// TIA Portal V19 export
FUNCTION "FC_EM_Loading" : Void   // FC3, FBD
{ S7_Optimized_Access := 'TRUE' }
// stored: SetENOAutomatically false
BEGIN

REGION Network 1: ------------------------------------------------------------------------ Inputs ------------------------------------------------------------------------
END_REGION

REGION Network 2: Verwerken iLoadingSenDown_a1
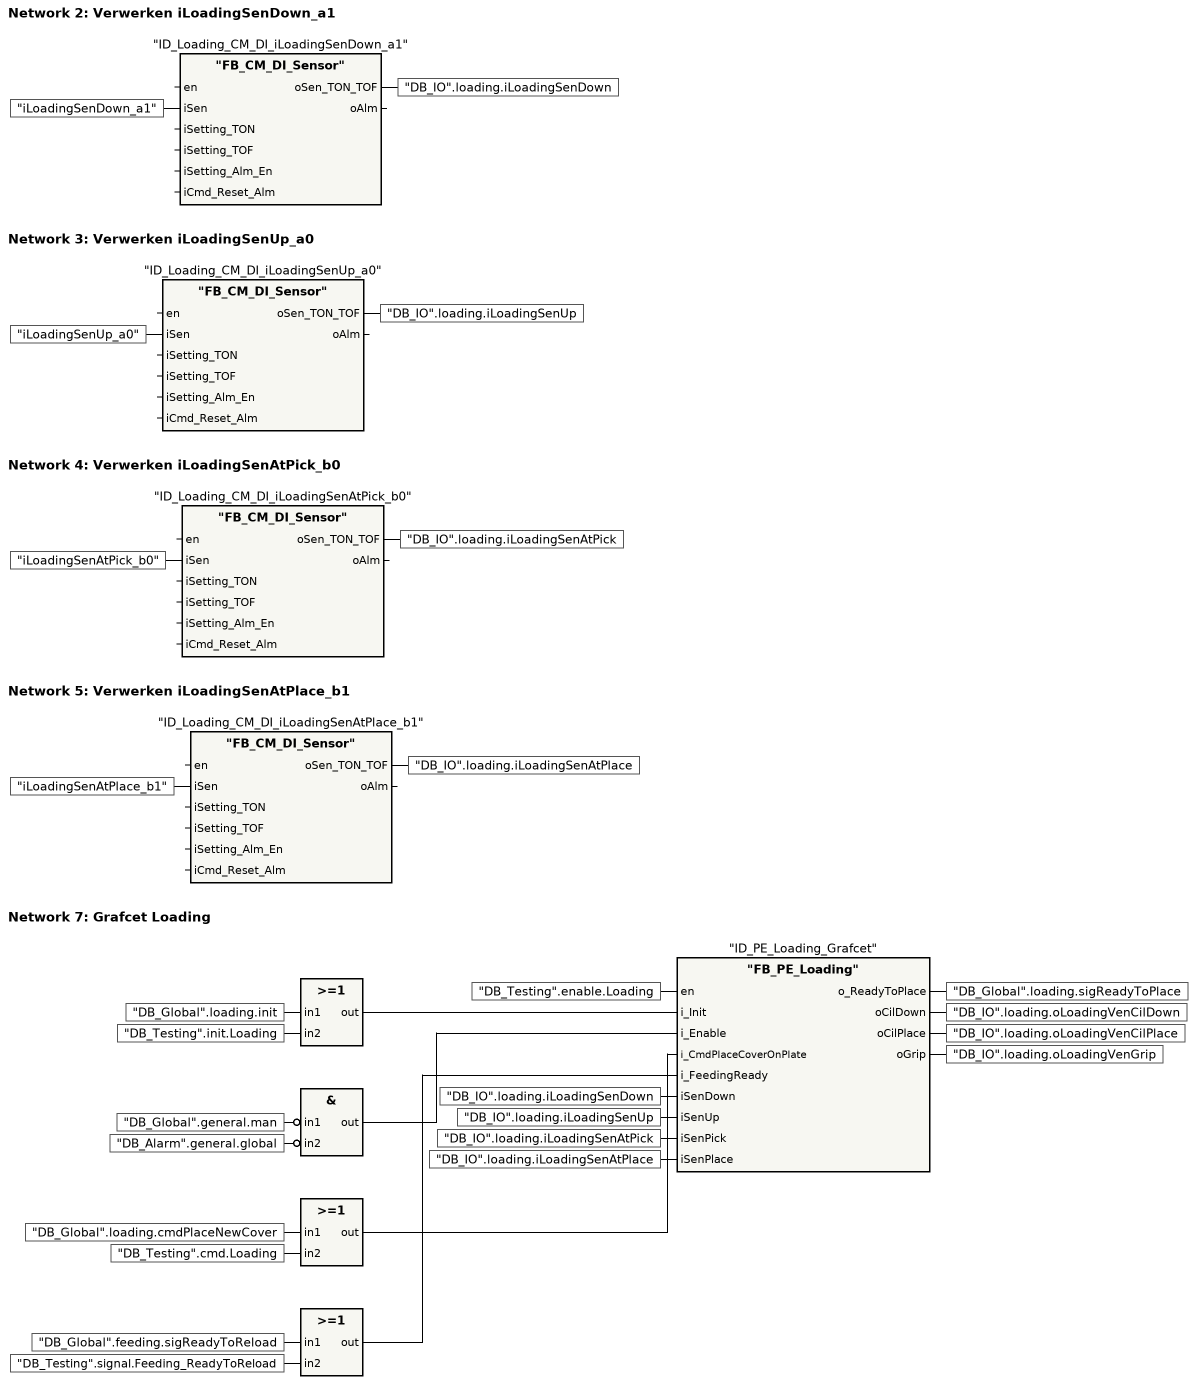
   "ID_Loading_CM_DI_iLoadingSenDown_a1"(iSen := "iLoadingSenDown_a1",   // "FB_CM_DI_Sensor"
                           oSen_TON_TOF => "DB_IO".loading.iLoadingSenDown);
END_REGION

REGION Network 3: Verwerken iLoadingSenUp_a0
   "ID_Loading_CM_DI_iLoadingSenUp_a0"(iSen := "iLoadingSenUp_a0",   // "FB_CM_DI_Sensor"
                           oSen_TON_TOF => "DB_IO".loading.iLoadingSenUp);
END_REGION

REGION Network 4: Verwerken iLoadingSenAtPick_b0
   "ID_Loading_CM_DI_iLoadingSenAtPick_b0"(iSen := "iLoadingSenAtPick_b0",   // "FB_CM_DI_Sensor"
                           oSen_TON_TOF => "DB_IO".loading.iLoadingSenAtPick);
END_REGION

REGION Network 5: Verwerken iLoadingSenAtPlace_b1
   "ID_Loading_CM_DI_iLoadingSenAtPlace_b1"(iSen := "iLoadingSenAtPlace_b1",   // "FB_CM_DI_Sensor"
                           oSen_TON_TOF => "DB_IO".loading.iLoadingSenAtPlace);
END_REGION

REGION Network 6: ------------------------------------------------------------------------ Logic ------------------------------------------------------------------------
END_REGION

REGION Network 7: Grafcet Loading
   IF "DB_Testing".enable.Loading THEN
       "ID_PE_Loading_Grafcet"(i_Init := "DB_Global".loading.init OR "DB_Testing".init.Loading,   // "FB_PE_Loading"
                               i_Enable := NOT "DB_Global".general.man AND NOT "DB_Alarm".general.global,
                               i_CmdPlaceCoverOnPlate := "DB_Global".loading.cmdPlaceNewCover OR "DB_Testing".cmd.Loading,
                               i_FeedingReady := "DB_Global".feeding.sigReadyToReload OR "DB_Testing".signal.Feeding_ReadyToReload,
                               iSenDown := "DB_IO".loading.iLoadingSenDown,
                               iSenUp := "DB_IO".loading.iLoadingSenUp,
                               iSenPick := "DB_IO".loading.iLoadingSenAtPick,
                               iSenPlace := "DB_IO".loading.iLoadingSenAtPlace,
                               o_ReadyToPlace => "DB_Global".loading.sigReadyToPlace,
                               oCilDown => "DB_IO".loading.oLoadingVenCilDown,
                               oCilPlace => "DB_IO".loading.oLoadingVenCilPlace,
                               oGrip => "DB_IO".loading.oLoadingVenGrip);
   END_IF;
END_REGION

REGION Network 8: ------------------------------------------------------------------------ Outputs ------------------------------------------------------------------------
END_REGION

REGION Network 9: Sturen oLoadingVenCilDown_A+
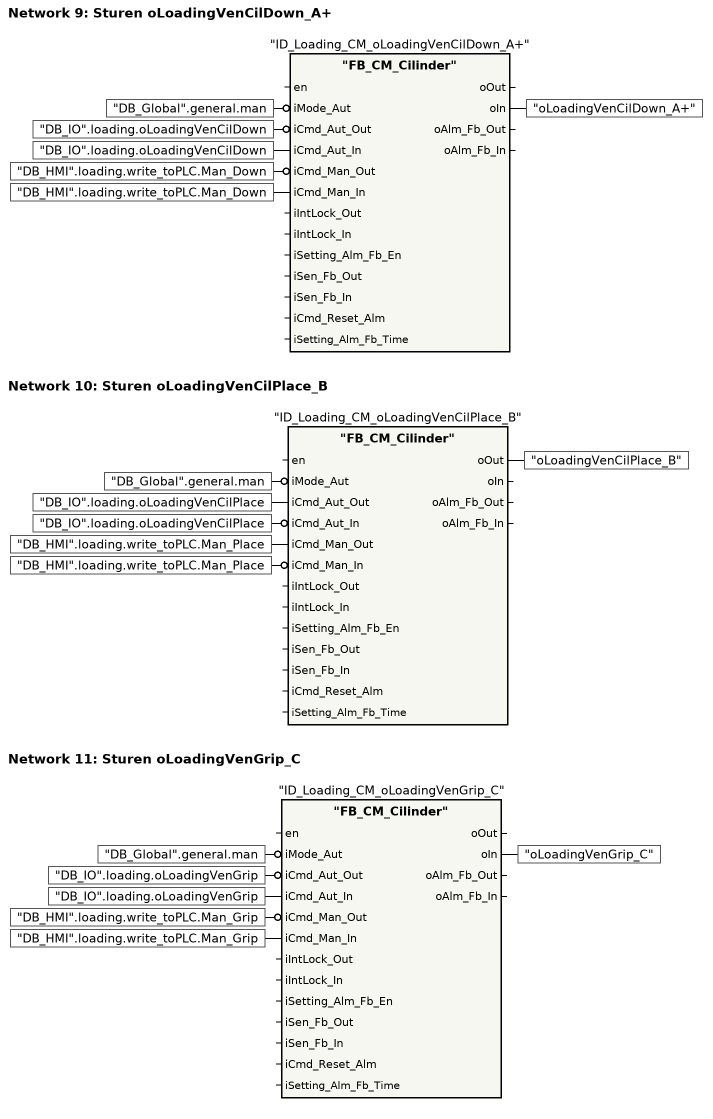
   "ID_Loading_CM_oLoadingVenCilDown_A+"(iMode_Aut := NOT "DB_Global".general.man,   // "FB_CM_Cilinder"
                           iCmd_Aut_Out := NOT "DB_IO".loading.oLoadingVenCilDown,
                           iCmd_Aut_In := "DB_IO".loading.oLoadingVenCilDown,
                           iCmd_Man_Out := NOT "DB_HMI".loading.write_toPLC.Man_Down,
                           iCmd_Man_In := "DB_HMI".loading.write_toPLC.Man_Down,
                           oIn => "oLoadingVenCilDown_A+");
END_REGION

REGION Network 10: Sturen oLoadingVenCilPlace_B
   "ID_Loading_CM_oLoadingVenCilPlace_B"(iMode_Aut := NOT "DB_Global".general.man,   // "FB_CM_Cilinder"
                           iCmd_Aut_Out := "DB_IO".loading.oLoadingVenCilPlace,
                           iCmd_Aut_In := NOT "DB_IO".loading.oLoadingVenCilPlace,
                           iCmd_Man_Out := "DB_HMI".loading.write_toPLC.Man_Place,
                           iCmd_Man_In := NOT "DB_HMI".loading.write_toPLC.Man_Place,
                           oOut => "oLoadingVenCilPlace_B");
END_REGION

REGION Network 11: Sturen oLoadingVenGrip_C
   "ID_Loading_CM_oLoadingVenGrip_C"(iMode_Aut := NOT "DB_Global".general.man,   // "FB_CM_Cilinder"
                           iCmd_Aut_Out := NOT "DB_IO".loading.oLoadingVenGrip,
                           iCmd_Aut_In := "DB_IO".loading.oLoadingVenGrip,
                           iCmd_Man_Out := NOT "DB_HMI".loading.write_toPLC.Man_Grip,
                           iCmd_Man_In := "DB_HMI".loading.write_toPLC.Man_Grip,
                           oIn => "oLoadingVenGrip_C");
END_REGION
END_FUNCTION
